// TIA Portal V20 export
DATA_BLOCK "DB_IO_Device_In_Functional_Test"   // DB6
{ S7_Optimized_Access := 'TRUE' }
// stored: MemoryReserve 100
   VAR
      Reset_PLC_Functional_Test : Array[0..31] of Bool;
      Status : Bool;
      Voltage_Read : UInt;
   END_VAR
BEGIN
END_DATA_BLOCK
